// TwinCAT 3 PLC project Machine
// ProgramVersion: 3.1.4022.1
// libraries:
//   GWP Library, * (Viessmann)
//   Tc2_Standard, * (Beckhoff Automation GmbH)
//   Tc2_System, * (Beckhoff Automation GmbH)
//   Tc2_Utilities, * (Beckhoff Automation GmbH)
//   Tc3_Module, * (Beckhoff Automation GmbH)
//   VisuDialogs, * (System)
//   VisuSymbols,3.5.10.0,System
// project tree:
//   / GlobalTextList.TcGTLO, PlcTask.TcTTO, Visualization Manager.TcVMO (not stored), VISU_TASK.TcTTO
//   POUs/ IOs.TcPOU, MAIN.TcPOU
//   VISUs/ Login.TcVIS, Fusszeile.TcVIS, Kreis.TcVIS, Home.TcVIS, EG.TcVIS, Menue.TcVIS, VD.TcVIS, KD.TcVIS, Alarmliste.TcVIS
// real-time tasks:
//   TASK PlcTask: cycle T#10ms, priority 20, ADS port 350
//   TASK VISU_TASK: cycle T#200000us, priority 30, ADS port 351
// I/O:
//   DEVICE Device 1 (EtherCAT), AmsNetId 5.49.104.148.2.1
//     Term 11 (EK1100) [EK1100 EtherCAT Coupler (2A E-Bus)]
//       Term 12 (EL1809) [EL1809 16Ch. Dig. Input 24V, 3ms]
//       Term 13 (EL2809) [EL2809 16Ch. Dig. Output 24V, 0.5A]
//       Term 14 (EL3208) [EL3208 8Ch. Ana. Input PT100 (RTD)]
//       Term 15 (EL3208) [EL3208 8Ch. Ana. Input PT100 (RTD)]
//       Term 16 (EL3058) [EL3058 8Ch. Ana. Input 4-20mA]
//       Term 17 (EL4008) [EL4008 8Ch. Ana. Output 0-10V, 12bit]
//       Term 18 (EL7031) [EL7031 1Ch. Stepper motor output stage (24V, 1.5A)]
//       Term 19 (EL9011) [EL9011 End Terminal]
// variable links:
//   Machine/Machine Instance <-> Device 1 (EtherCAT)/Term 11 (EK1100)/Term 12 (EL1809)
//     PlcTask Inputs/MAIN.IOs_0.DI_850KF2.ix_DI{1..16} <-> Channel {1..16}/Input  (16 links)
//   Machine/Machine Instance <-> Device 1 (EtherCAT)/Term 11 (EK1100)/Term 13 (EL2809)
//     PlcTask Outputs/MAIN.IOs_0.DO_850KF3.qx_DO{1..16} <-> Channel {1..16}/Output  (16 links)
//   Machine/Machine Instance <-> Device 1 (EtherCAT)/Term 11 (EK1100)/Term 14 (EL3208)
//     PlcTask Inputs/MAIN.IOs_0.AI_850KF4.ii_AI{1..8} <-> RTD Inputs Channel {1..8}/Value  (8 links)
//   Machine/Machine Instance <-> Device 1 (EtherCAT)/Term 11 (EK1100)/Term 15 (EL3208)
//     PlcTask Inputs/MAIN.IOs_0.AI_850KF4_1.ii_AI{1..8} <-> RTD Inputs Channel {1..8}/Value  (8 links)
//   Machine/Machine Instance <-> Device 1 (EtherCAT)/Term 11 (EK1100)/Term 16 (EL3058)
//     PlcTask Inputs/MAIN.IOs_0.AI_850KF5.ii_AI{1..8} <-> AI Standard Channel {1..8}/Value  (8 links)
//   Machine/Machine Instance <-> Device 1 (EtherCAT)/Term 11 (EK1100)/Term 17 (EL4008)
//     PlcTask Outputs/MAIN.IOs_0.AO_850KF6.qi_AO{1..8} <-> AO Outputs Channel {1..8}/Analog output  (8 links)
//   Machine/Machine Instance <-> Device 1 (EtherCAT)/Term 11 (EK1100)/Term 18 (EL7031)
//     PlcTask Inputs/MAIN.IOs_0.SM_850KF6_1.ii_CounterValue <-> ENC Status/Counter value
//     PlcTask Outputs/MAIN.IOs_0.SM_850KF6_1.qi_SetCounter <-> ENC Control/Set counter value
//     PlcTask Outputs/MAIN.IOs_0.SM_850KF6_1.qi_Velo <-> STM Velocity/Velocity
//     PlcTask Outputs/MAIN.IOs_0.SM_850KF6_1.qx_EN <-> STM Control/Control/Enable
//     PlcTask Outputs/MAIN.IOs_0.SM_850KF6_1.qx_SetCounter <-> ENC Control/Control/Set counter

CONFIGURATION Machine
    RESOURCE PLC ON TwinCAT3
        TASK PlcTask(INTERVAL := T#10ms, PRIORITY := 20);
        TASK VISU_TASK(INTERVAL := T#200000us, PRIORITY := 30);
        PROGRAM MAIN WITH PlcTask : MAIN;
        PROGRAM VisuElems_Visu_Prg WITH VISU_TASK : VisuElems.Visu_Prg;
    END_RESOURCE
END_CONFIGURATION

// ---- POUs/MAIN.TcPOU
PROGRAM MAIN
VAR PERSISTENT
	SW_Liste:SW_Struct;
END_VAR
VAR
	VD_0: VD;
	Kreis_3KO_0: Kreis_3KO;
	KD_0: KD;
	IOs_0: IOs;
	AI_to_Druck_0: AI_to_Druck;
	AI_to_Druck_1: AI_to_Druck;
	Init_0: Init;
	i_anzahlStufen: INT;
	einestufe: BOOL;
	zweitestufe: BOOL;
	Logger_0: logger;
	COUNT_0: count;
	Alarme_1bis10: alarm;
	Alarme_11bis20: alarm;
	Alarme_21bis30: alarm;
END_VAR

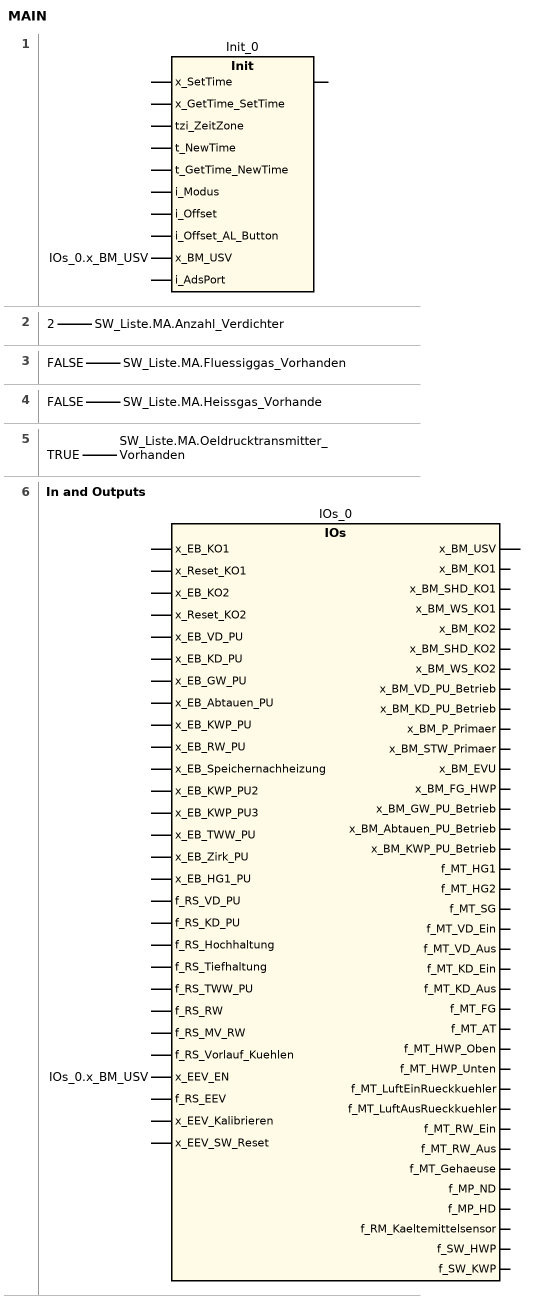
// NETWORK 1
Init_0(x_BM_USV := IOs_0.x_BM_USV); // Init

// NETWORK 2
SW_Liste.MA.Anzahl_Verdichter := 2;

// NETWORK 3
SW_Liste.MA.Fluessiggas_Vorhanden := FALSE;

// NETWORK 4
SW_Liste.MA.Heissgas_Vorhande := FALSE;

// NETWORK 5
SW_Liste.MA.Oeldrucktransmitter_Vorhanden := TRUE;

// NETWORK 6: In and Outputs
IOs_0(x_EEV_EN := IOs_0.x_BM_USV); // IOs

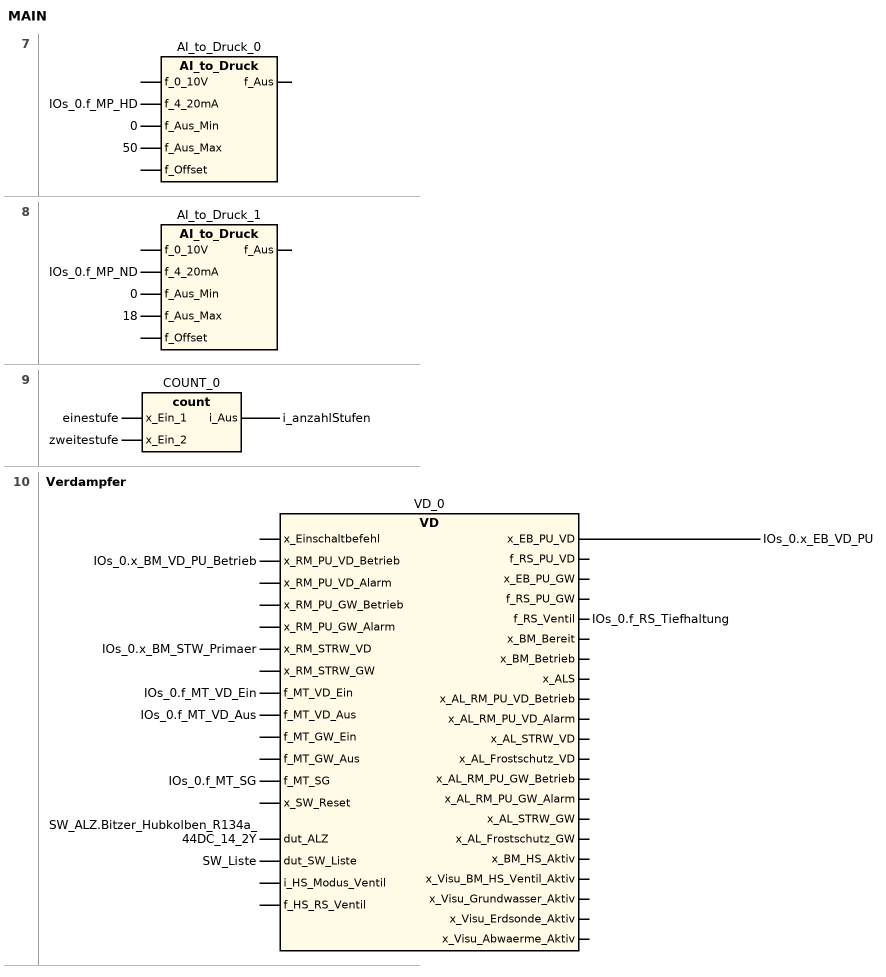
// NETWORK 7
AI_to_Druck_0(f_4_20mA := IOs_0.f_MP_HD, f_Aus_Min := 0, f_Aus_Max := 50); // AI_to_Druck

// NETWORK 8
AI_to_Druck_1(f_4_20mA := IOs_0.f_MP_ND, f_Aus_Min := 0, f_Aus_Max := 18); // AI_to_Druck

// NETWORK 9
COUNT_0(x_Ein_1 := einestufe, x_Ein_2 := zweitestufe); // count
i_anzahlStufen := COUNT_0.i_Aus;

// NETWORK 10: Verdampfer
VD_0(
    x_RM_PU_VD_Betrieb := IOs_0.x_BM_VD_PU_Betrieb,
    x_RM_STRW_VD := IOs_0.x_BM_STW_Primaer,
    f_MT_VD_Ein := IOs_0.f_MT_VD_Ein,
    f_MT_VD_Aus := IOs_0.f_MT_VD_Aus,
    f_MT_SG := IOs_0.f_MT_SG,
    dut_ALZ := SW_ALZ.Bitzer_Hubkolben_R134a_44DC_14_2Y,
    dut_SW_Liste := SW_Liste,
    f_RS_Ventil => IOs_0.f_RS_Tiefhaltung); // VD
IOs_0.x_EB_VD_PU := VD_0.x_EB_PU_VD;

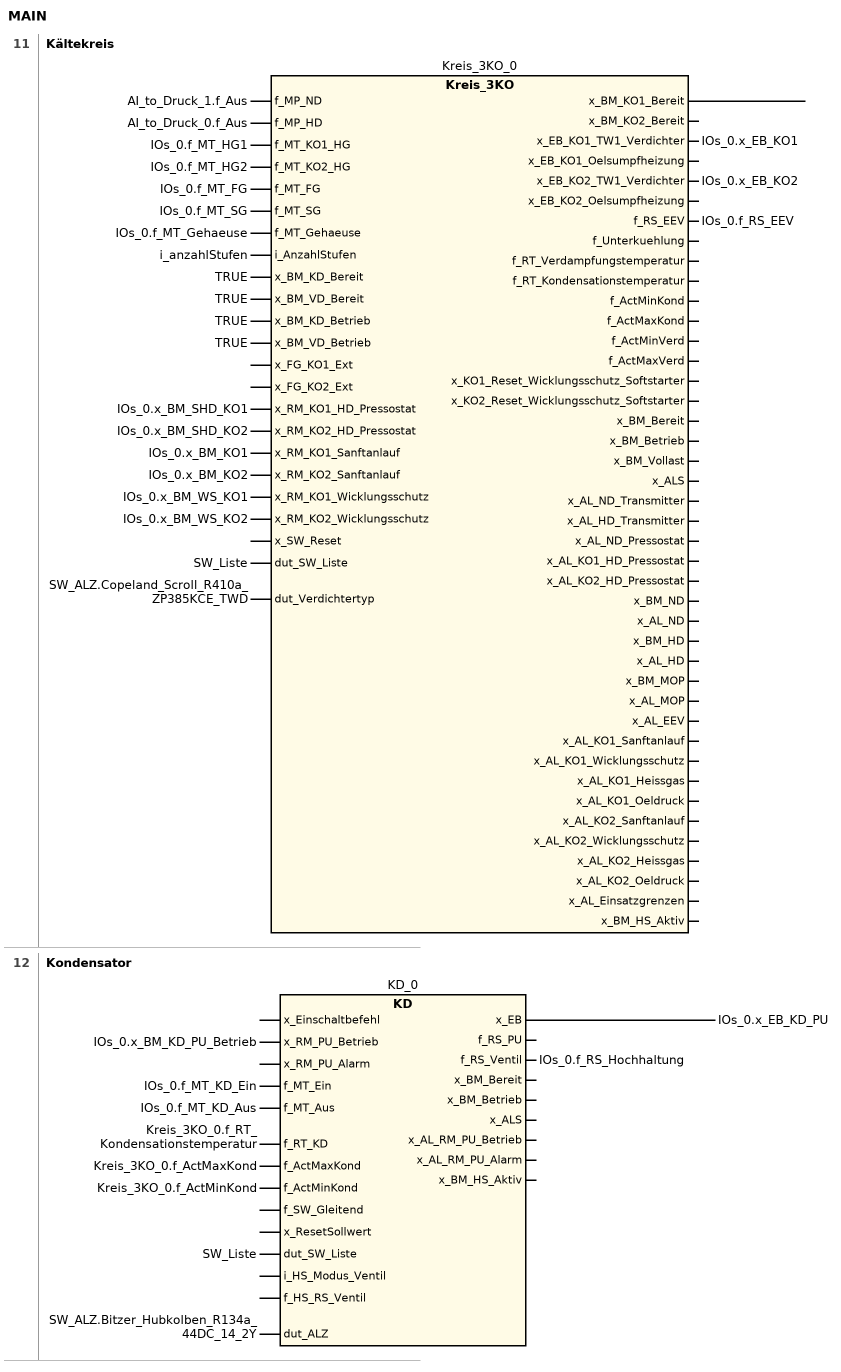
// NETWORK 11: Kältekreis
Kreis_3KO_0(
    f_MP_ND := AI_to_Druck_1.f_Aus,
    f_MP_HD := AI_to_Druck_0.f_Aus,
    f_MT_KO1_HG := IOs_0.f_MT_HG1,
    f_MT_KO2_HG := IOs_0.f_MT_HG2,
    f_MT_FG := IOs_0.f_MT_FG,
    f_MT_SG := IOs_0.f_MT_SG,
    f_MT_Gehaeuse := IOs_0.f_MT_Gehaeuse,
    i_AnzahlStufen := i_anzahlStufen,
    x_BM_KD_Bereit := TRUE,
    x_BM_VD_Bereit := TRUE,
    x_BM_KD_Betrieb := TRUE,
    x_BM_VD_Betrieb := TRUE,
    x_RM_KO1_HD_Pressostat := IOs_0.x_BM_SHD_KO1,
    x_RM_KO2_HD_Pressostat := IOs_0.x_BM_SHD_KO2,
    x_RM_KO1_Sanftanlauf := IOs_0.x_BM_KO1,
    x_RM_KO2_Sanftanlauf := IOs_0.x_BM_KO2,
    x_RM_KO1_Wicklungsschutz := IOs_0.x_BM_WS_KO1,
    x_RM_KO2_Wicklungsschutz := IOs_0.x_BM_WS_KO2,
    dut_SW_Liste := SW_Liste,
    dut_Verdichtertyp := SW_ALZ.Copeland_Scroll_R410a_ZP385KCE_TWD,
    x_EB_KO1_TW1_Verdichter => IOs_0.x_EB_KO1,
    x_EB_KO2_TW1_Verdichter => IOs_0.x_EB_KO2,
    f_RS_EEV => IOs_0.f_RS_EEV); // Kreis_3KO

// NETWORK 12: Kondensator
KD_0(
    x_RM_PU_Betrieb := IOs_0.x_BM_KD_PU_Betrieb,
    f_MT_Ein := IOs_0.f_MT_KD_Ein,
    f_MT_Aus := IOs_0.f_MT_KD_Aus,
    f_RT_KD := Kreis_3KO_0.f_RT_Kondensationstemperatur,
    f_ActMaxKond := Kreis_3KO_0.f_ActMaxKond,
    f_ActMinKond := Kreis_3KO_0.f_ActMinKond,
    dut_SW_Liste := SW_Liste,
    dut_ALZ := SW_ALZ.Bitzer_Hubkolben_R134a_44DC_14_2Y,
    f_RS_Ventil => IOs_0.f_RS_Hochhaltung); // KD
IOs_0.x_EB_KD_PU := KD_0.x_EB;

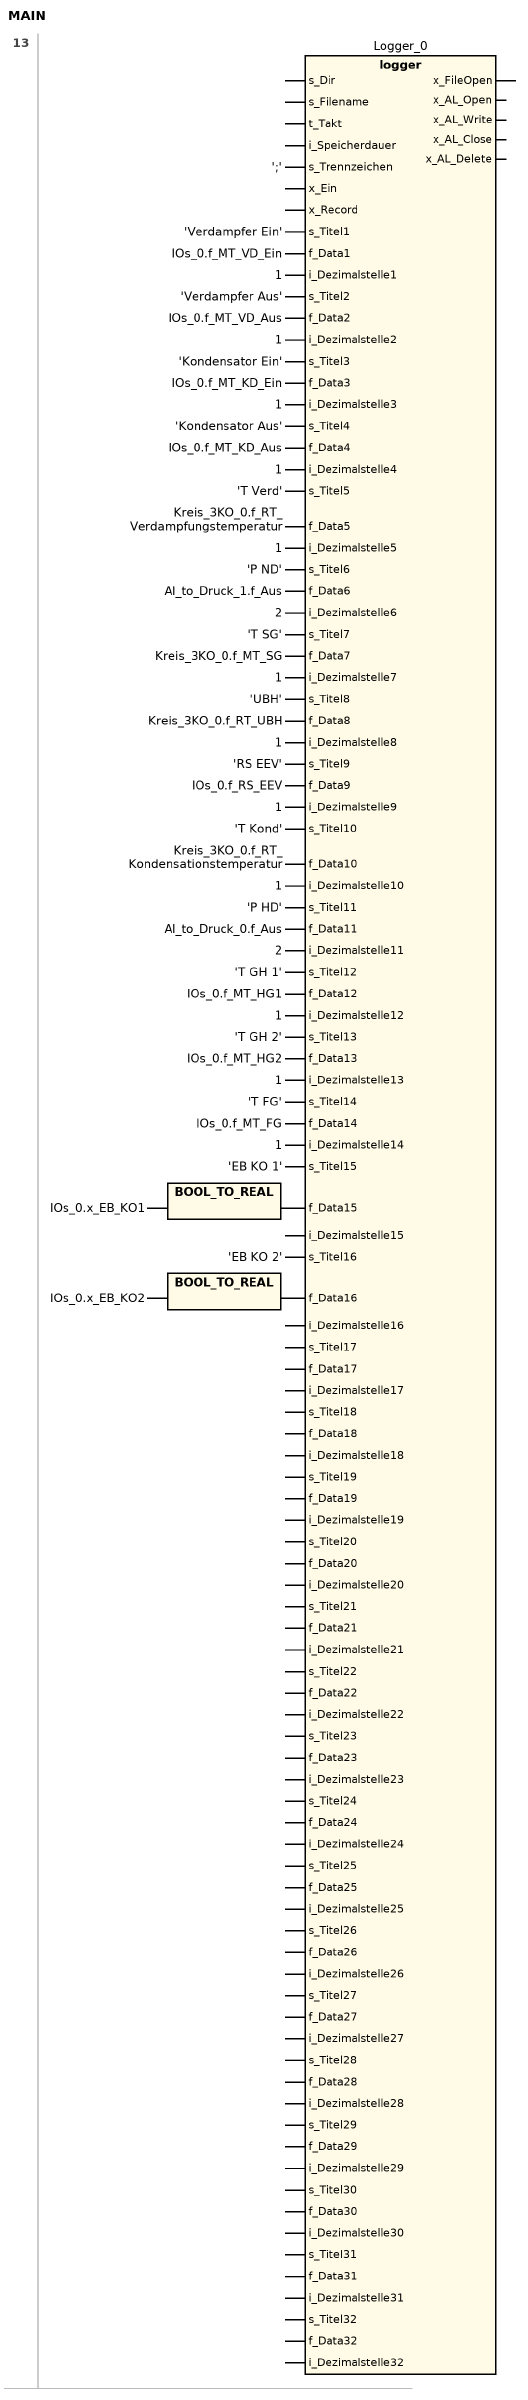
// NETWORK 13
Logger_0(
    s_Trennzeichen := ';',
    s_Titel1 := 'Verdampfer Ein',
    f_Data1 := IOs_0.f_MT_VD_Ein,
    i_Dezimalstelle1 := 1,
    s_Titel2 := 'Verdampfer Aus',
    f_Data2 := IOs_0.f_MT_VD_Aus,
    i_Dezimalstelle2 := 1,
    s_Titel3 := 'Kondensator Ein',
    f_Data3 := IOs_0.f_MT_KD_Ein,
    i_Dezimalstelle3 := 1,
    s_Titel4 := 'Kondensator Aus',
    f_Data4 := IOs_0.f_MT_KD_Aus,
    i_Dezimalstelle4 := 1,
    s_Titel5 := 'T Verd',
    f_Data5 := Kreis_3KO_0.f_RT_Verdampfungstemperatur,
    i_Dezimalstelle5 := 1,
    s_Titel6 := 'P ND',
    f_Data6 := AI_to_Druck_1.f_Aus,
    i_Dezimalstelle6 := 2,
    s_Titel7 := 'T SG',
    f_Data7 := Kreis_3KO_0.f_MT_SG,
    i_Dezimalstelle7 := 1,
    s_Titel8 := 'UBH',
    f_Data8 := Kreis_3KO_0.f_RT_UBH,
    i_Dezimalstelle8 := 1,
    s_Titel9 := 'RS EEV',
    f_Data9 := IOs_0.f_RS_EEV,
    i_Dezimalstelle9 := 1,
    s_Titel10 := 'T Kond',
    f_Data10 := Kreis_3KO_0.f_RT_Kondensationstemperatur,
    i_Dezimalstelle10 := 1,
    s_Titel11 := 'P HD',
    f_Data11 := AI_to_Druck_0.f_Aus,
    i_Dezimalstelle11 := 2,
    s_Titel12 := 'T GH 1',
    f_Data12 := IOs_0.f_MT_HG1,
    i_Dezimalstelle12 := 1,
    s_Titel13 := 'T GH 2',
    f_Data13 := IOs_0.f_MT_HG2,
    i_Dezimalstelle13 := 1,
    s_Titel14 := 'T FG',
    f_Data14 := IOs_0.f_MT_FG,
    i_Dezimalstelle14 := 1,
    s_Titel15 := 'EB KO 1',
    f_Data15 := BOOL_TO_REAL(IOs_0.x_EB_KO1),
    s_Titel16 := 'EB KO 2',
    f_Data16 := BOOL_TO_REAL(IOs_0.x_EB_KO2)); // logger

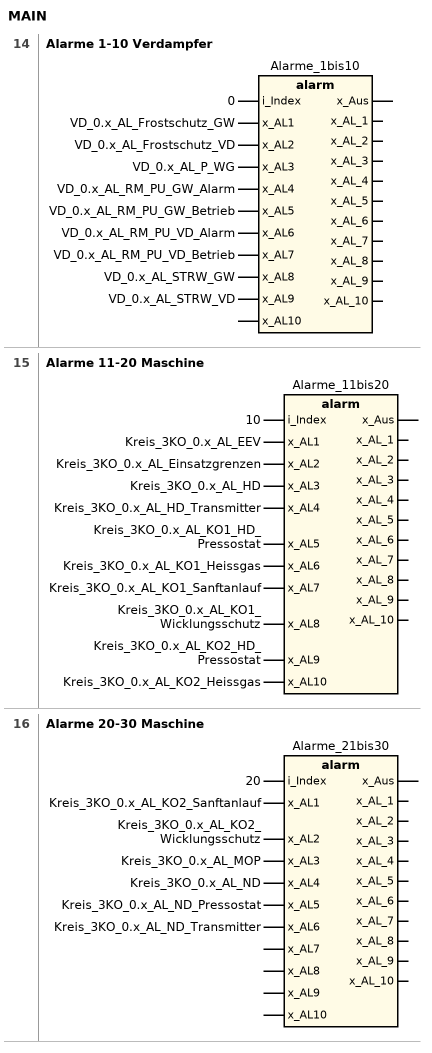
// NETWORK 14: Alarme 1-10 Verdampfer
Alarme_1bis10(
    i_Index := 0,
    x_AL1 := VD_0.x_AL_Frostschutz_GW,
    x_AL2 := VD_0.x_AL_Frostschutz_VD,
    x_AL3 := VD_0.x_AL_P_WG,
    x_AL4 := VD_0.x_AL_RM_PU_GW_Alarm,
    x_AL5 := VD_0.x_AL_RM_PU_GW_Betrieb,
    x_AL6 := VD_0.x_AL_RM_PU_VD_Alarm,
    x_AL7 := VD_0.x_AL_RM_PU_VD_Betrieb,
    x_AL8 := VD_0.x_AL_STRW_GW,
    x_AL9 := VD_0.x_AL_STRW_VD); // alarm

// NETWORK 15: Alarme 11-20 Maschine
Alarme_11bis20(
    i_Index := 10,
    x_AL1 := Kreis_3KO_0.x_AL_EEV,
    x_AL2 := Kreis_3KO_0.x_AL_Einsatzgrenzen,
    x_AL3 := Kreis_3KO_0.x_AL_HD,
    x_AL4 := Kreis_3KO_0.x_AL_HD_Transmitter,
    x_AL5 := Kreis_3KO_0.x_AL_KO1_HD_Pressostat,
    x_AL6 := Kreis_3KO_0.x_AL_KO1_Heissgas,
    x_AL7 := Kreis_3KO_0.x_AL_KO1_Sanftanlauf,
    x_AL8 := Kreis_3KO_0.x_AL_KO1_Wicklungsschutz,
    x_AL9 := Kreis_3KO_0.x_AL_KO2_HD_Pressostat,
    x_AL10 := Kreis_3KO_0.x_AL_KO2_Heissgas); // alarm

// NETWORK 16: Alarme 20-30 Maschine
Alarme_21bis30(
    i_Index := 20,
    x_AL1 := Kreis_3KO_0.x_AL_KO2_Sanftanlauf,
    x_AL2 := Kreis_3KO_0.x_AL_KO2_Wicklungsschutz,
    x_AL3 := Kreis_3KO_0.x_AL_MOP,
    x_AL4 := Kreis_3KO_0.x_AL_ND,
    x_AL5 := Kreis_3KO_0.x_AL_ND_Pressostat,
    x_AL6 := Kreis_3KO_0.x_AL_ND_Transmitter); // alarm

END_PROGRAM

// ---- POUs/IOs.TcPOU
FUNCTION_BLOCK IOs
VAR_INPUT
	//850KF3
	x_EB_KO1: BOOL;
	x_Reset_KO1: BOOL;
	x_EB_KO2: BOOL;
	x_Reset_KO2: BOOL;
	x_EB_VD_PU: BOOL;
	x_EB_KD_PU: BOOL;
	x_EB_GW_PU: BOOL;
	x_EB_Abtauen_PU: BOOL;
	x_EB_KWP_PU: BOOL;
	x_EB_RW_PU: BOOL;
	x_EB_Speichernachheizung: BOOL;
	x_EB_KWP_PU2: BOOL;
	x_EB_KWP_PU3: BOOL;
	x_EB_TWW_PU: BOOL;
	x_EB_Zirk_PU: BOOL;
	x_EB_HG1_PU: BOOL;
	//850KF6
	f_RS_VD_PU: REAL;
	f_RS_KD_PU: REAL;
	f_RS_Hochhaltung: REAL;
	f_RS_Tiefhaltung: REAL;
	f_RS_TWW_PU: REAL;
	f_RS_RW: REAL;
	f_RS_MV_RW: REAL;
	f_RS_Vorlauf_Kuehlen: REAL;
	//850KF6.1
	x_EEV_EN: BOOL;
	f_RS_EEV: REAL;
	x_EEV_Kalibrieren: BOOL;
	x_EEV_SW_Reset: BOOL;
	
END_VAR
VAR_OUTPUT
	//850KF2
	x_BM_USV: BOOL;
	x_BM_KO1: BOOL;
	x_BM_SHD_KO1: BOOL;
	x_BM_WS_KO1: BOOL;
	x_BM_KO2: BOOL;
	x_BM_SHD_KO2: BOOL;
	x_BM_WS_KO2: BOOL;
	x_BM_VD_PU_Betrieb: BOOL;
	x_BM_KD_PU_Betrieb: BOOL;
	x_BM_P_Primaer: BOOL;
	x_BM_STW_Primaer: BOOL;
	x_BM_EVU: BOOL;
	x_BM_FG_HWP: BOOL;
	x_BM_GW_PU_Betrieb: BOOL;
	x_BM_Abtauen_PU_Betrieb: BOOL;
	x_BM_KWP_PU_Betrieb: BOOL;
	//850KF4
	f_MT_HG1: REAL;
	f_MT_HG2: REAL;
	f_MT_SG: REAL;
	f_MT_VD_Ein: REAL;
	f_MT_VD_Aus: REAL;
	f_MT_KD_Ein: REAL;
	f_MT_KD_Aus: REAL;
	f_MT_FG: REAL;
	//850KF4.1
	f_MT_AT: REAL;
	f_MT_HWP_Oben: REAL;
	f_MT_HWP_Unten: REAL;
	f_MT_LuftEinRueckkuehler: REAL;
	f_MT_LuftAusRueckkuehler: REAL;
	f_MT_RW_Ein: REAL;
	f_MT_RW_Aus: REAL;
	f_MT_Gehaeuse: REAL;
	//850KF5
	f_MP_ND: REAL;
	f_MP_HD: REAL;
	f_RM_Kaeltemittelsensor: REAL;
	f_SW_HWP: REAL;
	f_SW_KWP: REAL;
END_VAR
VAR
	DI_850KF2: DI_16;
	DO_850KF3: DO_16;
	AI_850KF4: AI_8_Temp;
	AI_850KF4_1: AI_8_Temp;
	AI_850KF5: AI_8_4_20mA;
	AO_850KF6: AO_8;
	SM_850KF6_1: EEV_Schrittmotor;
	
END_VAR

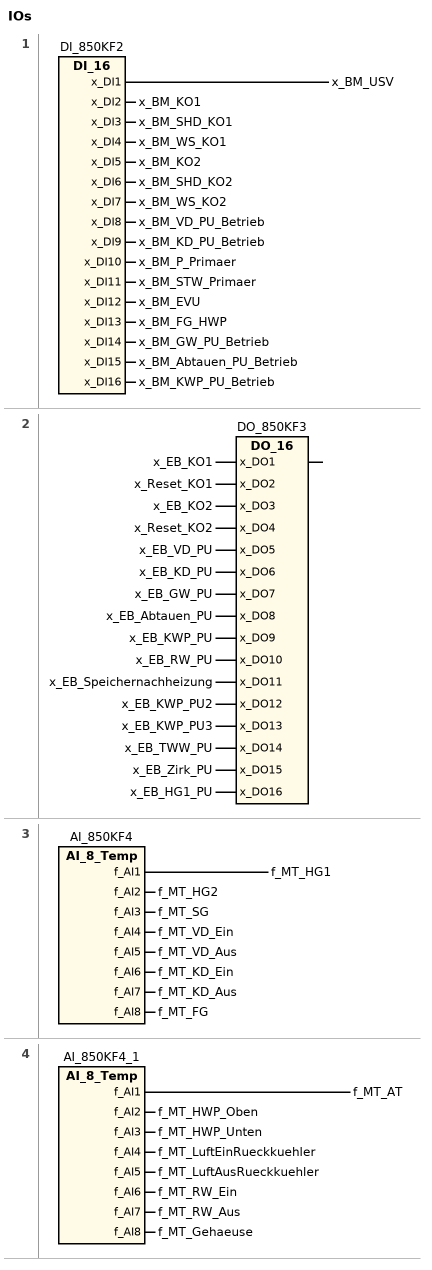
// NETWORK 1
DI_850KF2(
    x_DI2 => x_BM_KO1,
    x_DI3 => x_BM_SHD_KO1,
    x_DI4 => x_BM_WS_KO1,
    x_DI5 => x_BM_KO2,
    x_DI6 => x_BM_SHD_KO2,
    x_DI7 => x_BM_WS_KO2,
    x_DI8 => x_BM_VD_PU_Betrieb,
    x_DI9 => x_BM_KD_PU_Betrieb,
    x_DI10 => x_BM_P_Primaer,
    x_DI11 => x_BM_STW_Primaer,
    x_DI12 => x_BM_EVU,
    x_DI13 => x_BM_FG_HWP,
    x_DI14 => x_BM_GW_PU_Betrieb,
    x_DI15 => x_BM_Abtauen_PU_Betrieb,
    x_DI16 => x_BM_KWP_PU_Betrieb); // DI_16
x_BM_USV := DI_850KF2.x_DI1;

// NETWORK 2
DO_850KF3(
    x_DO1 := x_EB_KO1,
    x_DO2 := x_Reset_KO1,
    x_DO3 := x_EB_KO2,
    x_DO4 := x_Reset_KO2,
    x_DO5 := x_EB_VD_PU,
    x_DO6 := x_EB_KD_PU,
    x_DO7 := x_EB_GW_PU,
    x_DO8 := x_EB_Abtauen_PU,
    x_DO9 := x_EB_KWP_PU,
    x_DO10 := x_EB_RW_PU,
    x_DO11 := x_EB_Speichernachheizung,
    x_DO12 := x_EB_KWP_PU2,
    x_DO13 := x_EB_KWP_PU3,
    x_DO14 := x_EB_TWW_PU,
    x_DO15 := x_EB_Zirk_PU,
    x_DO16 := x_EB_HG1_PU); // DO_16

// NETWORK 3
AI_850KF4(
    f_AI2 => f_MT_HG2,
    f_AI3 => f_MT_SG,
    f_AI4 => f_MT_VD_Ein,
    f_AI5 => f_MT_VD_Aus,
    f_AI6 => f_MT_KD_Ein,
    f_AI7 => f_MT_KD_Aus,
    f_AI8 => f_MT_FG); // AI_8_Temp
f_MT_HG1 := AI_850KF4.f_AI1;

// NETWORK 4
AI_850KF4_1(
    f_AI2 => f_MT_HWP_Oben,
    f_AI3 => f_MT_HWP_Unten,
    f_AI4 => f_MT_LuftEinRueckkuehler,
    f_AI5 => f_MT_LuftAusRueckkuehler,
    f_AI6 => f_MT_RW_Ein,
    f_AI7 => f_MT_RW_Aus,
    f_AI8 => f_MT_Gehaeuse); // AI_8_Temp
f_MT_AT := AI_850KF4_1.f_AI1;

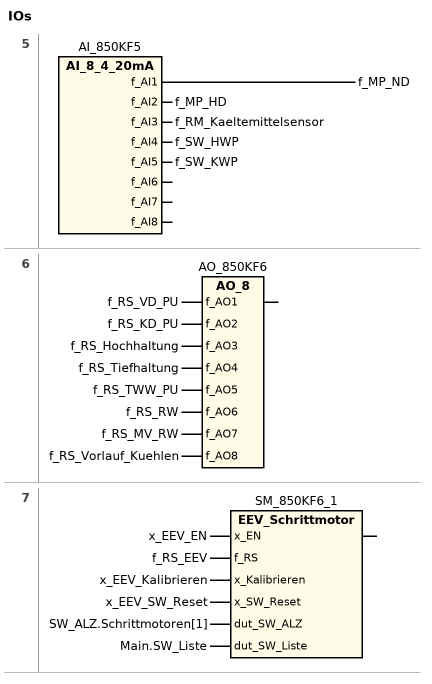
// NETWORK 5
AI_850KF5(f_AI2 => f_MP_HD, f_AI3 => f_RM_Kaeltemittelsensor, f_AI4 => f_SW_HWP, f_AI5 => f_SW_KWP); // AI_8_4_20mA
f_MP_ND := AI_850KF5.f_AI1;

// NETWORK 6
AO_850KF6(
    f_AO1 := f_RS_VD_PU,
    f_AO2 := f_RS_KD_PU,
    f_AO3 := f_RS_Hochhaltung,
    f_AO4 := f_RS_Tiefhaltung,
    f_AO5 := f_RS_TWW_PU,
    f_AO6 := f_RS_RW,
    f_AO7 := f_RS_MV_RW,
    f_AO8 := f_RS_Vorlauf_Kuehlen); // AO_8

// NETWORK 7
SM_850KF6_1(
    x_EN := x_EEV_EN,
    f_RS := f_RS_EEV,
    x_Kalibrieren := x_EEV_Kalibrieren,
    x_SW_Reset := x_EEV_SW_Reset,
    dut_SW_ALZ := SW_ALZ.Schrittmotoren[1],
    dut_SW_Liste := Main.SW_Liste); // EEV_Schrittmotor

END_FUNCTION_BLOCK

// ---- GlobalTextList.TcGTLO
TEXTLIST GlobalTextList
  168 = 'Einsatzgrenzen'
  642 = 'Kalibrieren'
  362 = 'Quittieren'
END_TEXTLIST

// ---- VISUs/Login.TcVIS
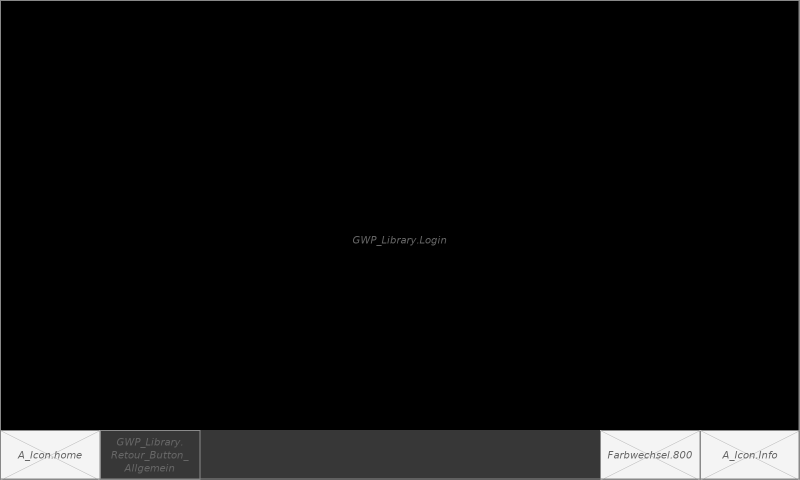
VISUALIZATION Login  // 800x480
    Frame (0,0 800x480)
        shows GWP_Library.Login()
    Frame (0,0 800x480)
        shows Fusszeile()
    Frame (100,430 100x50)
        shows GWP_Library.Retour_Button_Allgemein()
END_VISUALIZATION

// ---- VISUs/Fusszeile.TcVIS
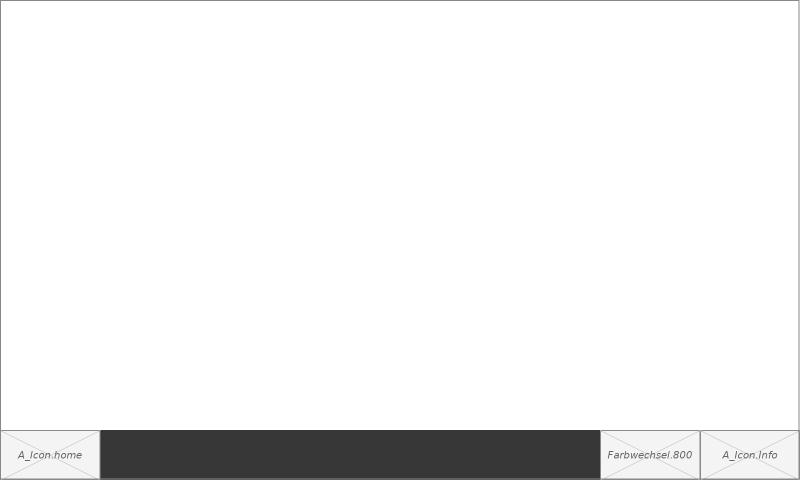
VISUALIZATION Fusszeile  // 800x480
    Rectangle (0,430 800x50)
    Image (600,430 100x50), image: Farbwechsel.800
        p84334746: Visu.s_Status_AL_Button
        OnMouseClick: change screen: Alarmliste
    Image (700,430 100x50), image: A_Icon.Info
    Image (0,430 100x50), image: A_Icon.home
        OnMouseClick: change screen: Home
END_VISUALIZATION

// ---- VISUs/Kreis.TcVIS
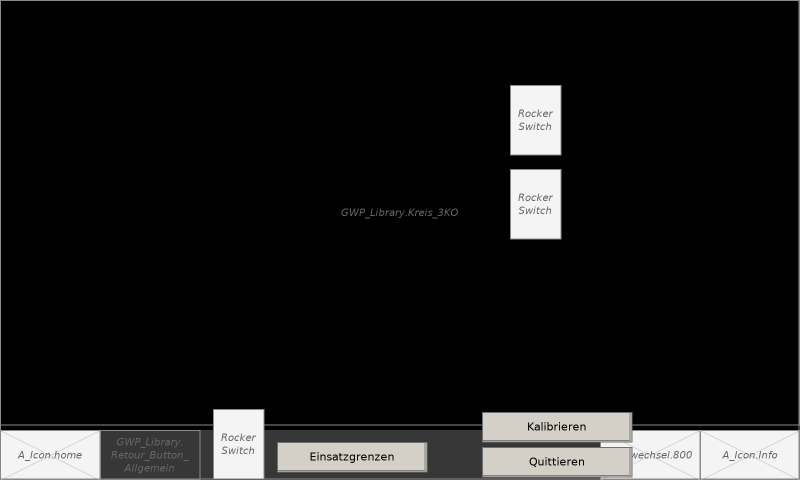
VISUALIZATION Kreis  // 800x480
    Frame (0,0 800x425)
        shows GWP_Library.Kreis_3KO(FB_Kreis_3KO := MAIN.Kreis_3KO_0, FB_KD := MAIN.KD_0, FB_VD := MAIN.VD_0)
    RockerSwitch (510,85 51x70), variable: MAIN.zweitestufe, behaviour: TOGGLE, style: Switch-RockerSwitch-Gray
    RockerSwitch (510,169 51x70), variable: MAIN.einestufe, behaviour: TOGGLE, style: Switch-RockerSwitch-Gray
    Frame (0,0 800x480)
        shows Fusszeile()
    Frame (100,430 100x50)
        shows GWP_Library.Retour_Button_Allgemein()
    RockerSwitch (213,409 51x70), variable: MAIN.Logger_0.x_Ein, behaviour: TOGGLE, style: Switch-RockerSwitch-Gray
    Button (277,442 150x30), "Einsatzgrenzen"
        OnMouseClick: change screen: EG
    Button (482,447 150x30), "Quittieren"
        tap GWP_Library.Globale_Variablen.x_Quittieren
    Button (482,412 150x30), "Kalibrieren"
        tap MAIN.IOs_0.x_EEV_Kalibrieren
END_VISUALIZATION

// ---- VISUs/Home.TcVIS
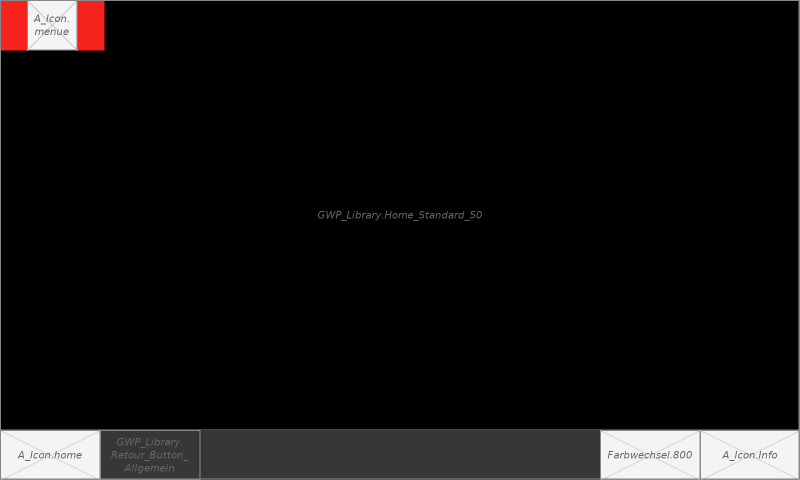
VISUALIZATION Home  // 800x480
    Frame (0,0 800x430)
        shows GWP_Library.Home_Standard_50(fb_Init_1 := MAIN.Init_0)
    Frame (0,0 800x480)
        shows Fusszeile()
    Frame (100,430 100x50)
        shows GWP_Library.Retour_Button_Allgemein()
    Group (0,0 104x50)
        OnMouseClick: change screen: Menue
        Rectangle (0,0 104x50)
        Image (27,0 50x50), image: A_Icon.menue
END_VISUALIZATION

// ---- VISUs/EG.TcVIS
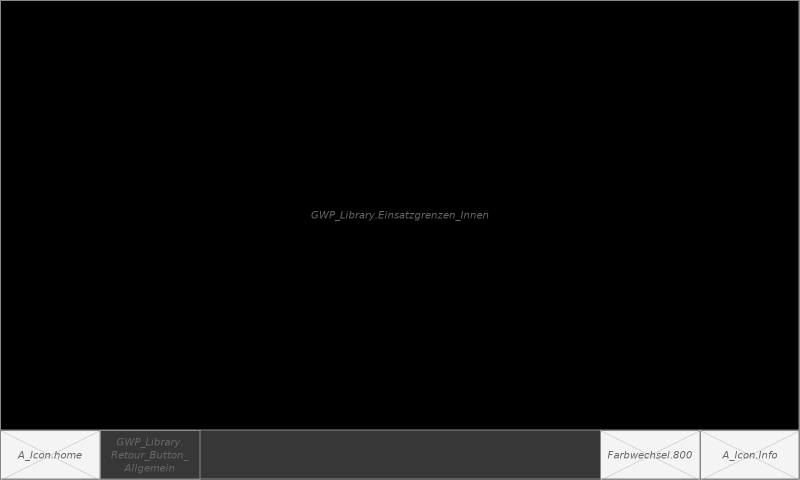
VISUALIZATION EG  // 800x480
    Frame (0,0 800x480)
        shows Fusszeile()
    Frame (100,430 100x50)
        shows GWP_Library.Retour_Button_Allgemein()
    Frame (0,0 800x430)
        shows GWP_Library.Einsatzgrenzen_Innen(FB_Einsatzgrenzen_Innen := MAIN.Kreis_3KO_0.Einsatzgrenzen_Innen)
END_VISUALIZATION

// ---- VISUs/Menue.TcVIS
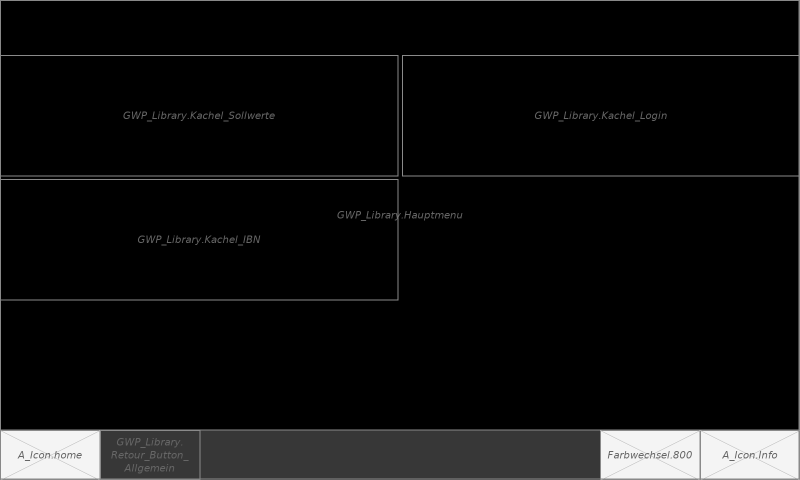
VISUALIZATION Menue  // 800x480
    Frame (0,0 800x480)
        shows Fusszeile()
    Frame (100,430 100x50)
        shows GWP_Library.Retour_Button_Allgemein()
    Frame (0,0 800x430)
        shows GWP_Library.Hauptmenu()
    Frame (0,55 398x121)
        shows GWP_Library.Kachel_Sollwerte()
        OnMouseClick: change screen: Sollwertmenu
    Frame (402,55 398x121)
        shows GWP_Library.Kachel_Login()
        OnMouseClick: change screen: Login
    Frame (0,179 398x121)
        shows GWP_Library.Kachel_IBN()
        OnMouseClick: change screen: IBS_Menu
END_VISUALIZATION

// ---- VISUs/VD.TcVIS
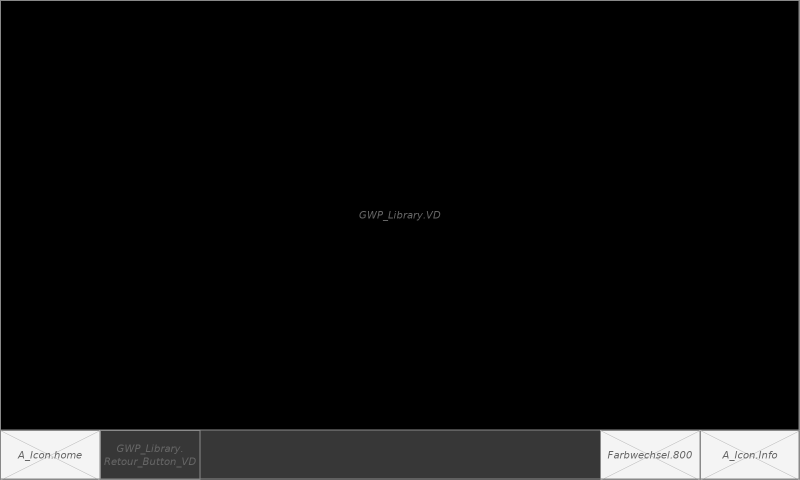
VISUALIZATION VD  // 800x480
    Frame (0,0 800x480)
        shows Fusszeile()
    Frame (100,430 100x50)
        shows GWP_Library.Retour_Button_VD()
    Frame (0,0 800x430)
        shows GWP_Library.VD(FB_VD := MAIN.VD_0)
END_VISUALIZATION

// ---- VISUs/KD.TcVIS
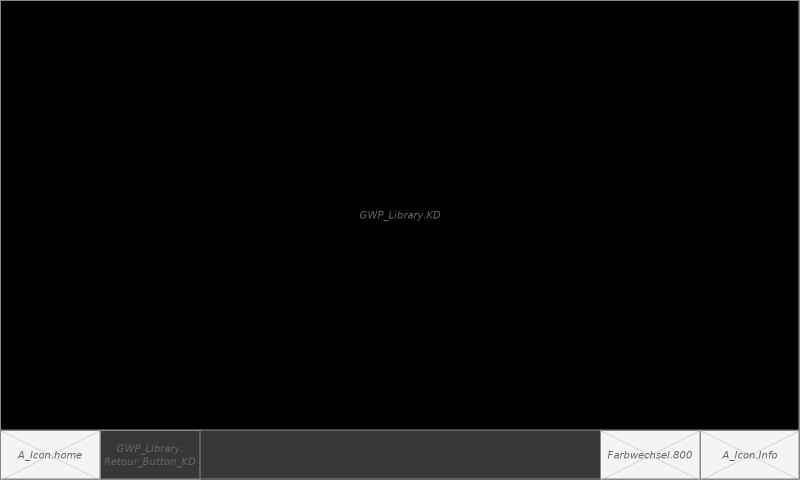
VISUALIZATION KD  // 800x480
    Frame (0,0 800x480)
        shows Fusszeile()
    Frame (100,430 100x50)
        shows GWP_Library.Retour_Button_KD()
    Frame (0,0 800x430)
        shows GWP_Library.KD(FB_KD := MAIN.KD_0)
END_VISUALIZATION

// ---- VISUs/Alarmliste.TcVIS
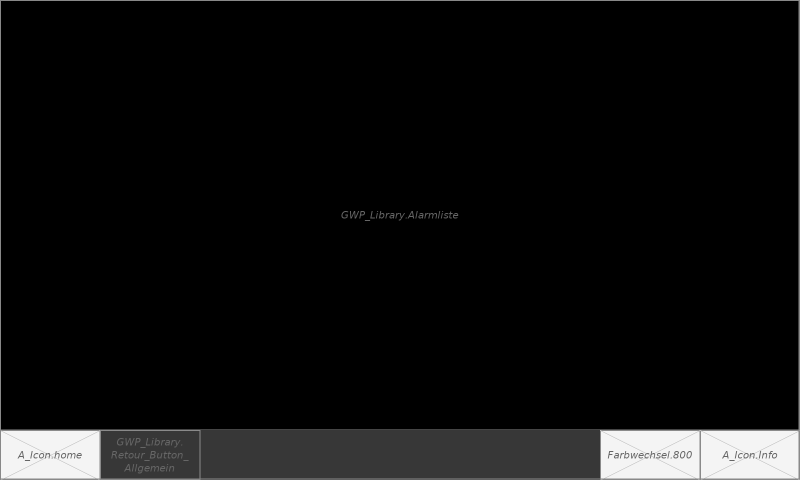
VISUALIZATION Alarmliste  // 800x480
    Frame (0,0 800x430)
        shows GWP_Library.Alarmliste()
    Frame (0,0 800x480)
        shows Fusszeile()
    Frame (100,430 100x50)
        shows GWP_Library.Retour_Button_Allgemein()
END_VISUALIZATION
